FUNCTION Convert_SINT_TO_UINT : Hresult
VAR_INPUT
	in : SINT;
	out : REFERENCE TO UINT;
END_VAR
VAR
	converted : UINT;
END_VAR
VAR CONSTANT
	INCOMPATIBLE : HRESULT := 16#9811070E;
END_VAR

converted := SINT_TO_UINT(in);

IF (UINT_TO_SINT(converted) <> in) THEN
	Convert_SINT_TO_UINT := INCOMPATIBLE;
	RETURN;
END_IF

out := converted;

END_FUNCTION

(* stored: Version 1.1.0.1, ProductVersion 3.1.4024.12
   POU Convert_SINT_TO_UINT: Id {e2c20f05-de01-4eee-ac96-459ebfcbee8f}, SpecialFunc None *)
